FUNCTION_BLOCK Incr
  (* Standard: 61499-2 *)
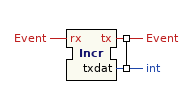
  EVENT_INPUT
    rx;
  END_EVENT
  EVENT_OUTPUT
    tx WITH txdat;
  END_EVENT
  VAR_OUTPUT
    txdat : int := 1;
  END_VAR
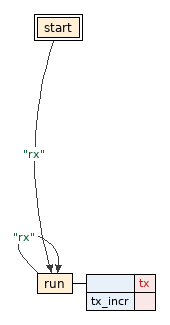
  EC_STATES
    start;
    run : -> tx, tx_incr;
  END_STATES
  EC_TRANSITIONS
    start TO run := "rx";
    run TO run := "rx";
  END_TRANSITIONS
  ALGORITHM tx_incr IN C:
me->txdat = me->txdat + 1;
  END_ALGORITHM
END_FUNCTION_BLOCK
